% RSLogix 500 project BINSCRUBBER #49 SETTON 9-12-2016 - copy Jeff.RSS, saved by version 10.00.00.00 %
PROJECT "JBT BIN"    % processor: MicroLogix 1200 %

PROGRAM FILES
  LAD 2 "MAIN"  10 rungs
  LAD 3 "START_UP"  7 rungs
  LAD 4 "ENCODER"  11 rungs
  LAD 5 "CRADDLE"  33 rungs
  LAD 6 "BRUSH"  26 rungs
  LAD 7 "WATER"  16 rungs
  LAD 8 "AUXILARY"  14 rungs
  LAD 9 "FAULTS"  43 rungs
  LAD 10 "CONVEYORS"  16 rungs
  LAD 11 "BIN SIZING"  9 rungs

DATA FILES
  O0 OUTPUT  6 elements
  I1 INPUT  6 elements
  S2 STATUS  66 elements
  B3 BINARY  5 elements
  T4 TIMER  35 elements
  C5 COUNTER  1 elements
  R6 CONTROL  1 elements
  N7 INTEGER  34 elements
  F8 FLOAT  1 elements
  L9   1 elements
  L10   2 elements

LADDER 2 "MAIN"
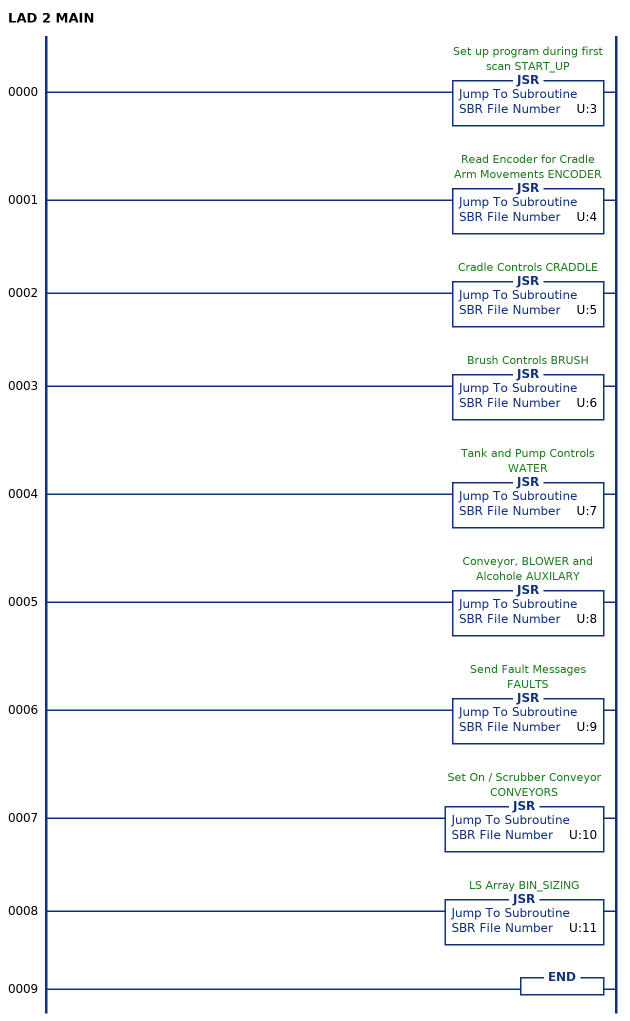
% Rung: 0 %
SOR JSR U:3 EOR
%   U:3  START_UP  "Set up program during first scan" %
% Rung: 1 %
SOR JSR U:4 EOR
%   U:4  ENCODER  "Read Encoder for Cradle Arm Movements" %
% Rung: 2 %
SOR JSR U:5 EOR
%   U:5  CRADDLE  "Cradle Controls" %
% Rung: 3 %
SOR JSR U:6 EOR
%   U:6  BRUSH  "Brush Controls" %
% Rung: 4 %
SOR JSR U:7 EOR
%   U:7  WATER  "Tank and Pump Controls" %
% Rung: 5 %
SOR JSR U:8 EOR
%   U:8  AUXILARY  "Conveyor, BLOWER and Alcohole" %
% Rung: 6 %
SOR JSR U:9 EOR
%   U:9  FAULTS  "Send Fault Messages" %
% Rung: 7 %
SOR JSR U:10 EOR
%   U:10  CONVEYORS  "Set On / Scrubber Conveyor" %
% Rung: 8 %
SOR JSR U:11 EOR
%   U:11  BIN_SIZING  "LS Array" %
% Rung: 9 %
SOR END EOR

LADDER 3 "START_UP"
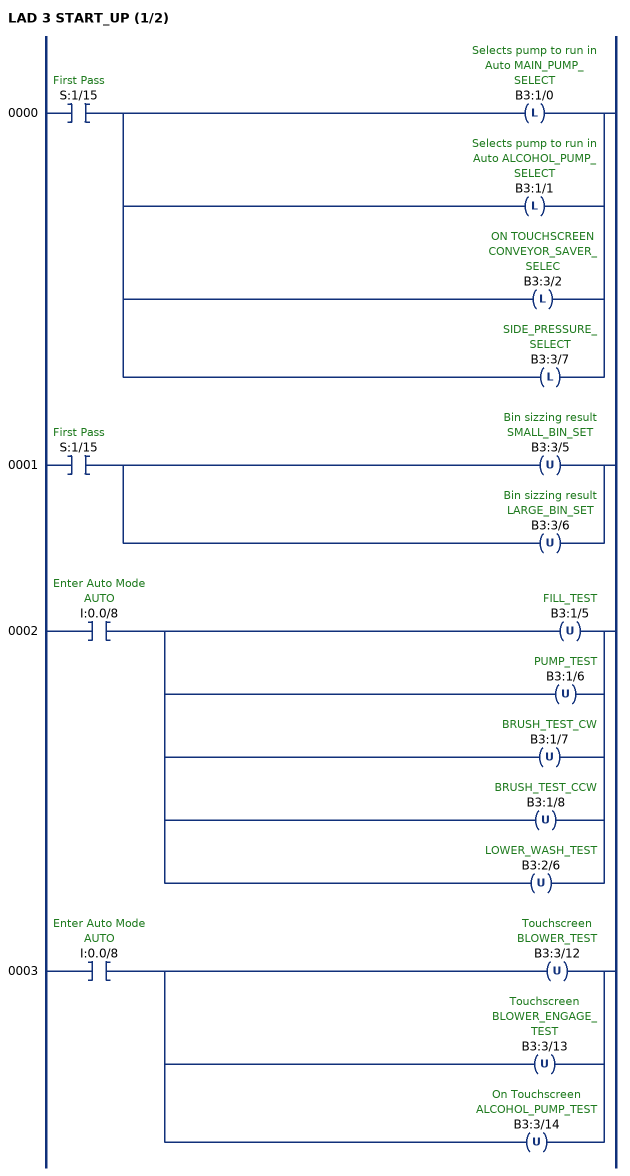
% Rung: 0 %
SOR XIC S:1/15 BST OTL B3:1/0 NXB BST OTL B3:1/1 NXB BST OTL B3:3/2 NXB OTL B3:3/7 BND BND BND EOR
%   S:1/15  "First Pass" %
%   B3:1/0  MAIN_PUMP_SELECT  "Selects pump to run in Auto" %
%   B3:1/1  ALCOHOL_PUMP_SELECT  "Selects pump to run in Auto" %
%   B3:3/2  CONVEYOR_SAVER_SELEC  "ON TOUCHSCREEN" %
%   B3:3/7  SIDE_PRESSURE_SELECT %
% Rung: 1 %
SOR XIC S:1/15 BST OTU B3:3/5 NXB OTU B3:3/6 BND EOR
%   S:1/15  "First Pass" %
%   B3:3/5  SMALL_BIN_SET  "Bin sizzing result" %
%   B3:3/6  LARGE_BIN_SET  "Bin sizzing result" %
% Rung: 2 %
SOR XIC I:0.0/8 BST OTU B3:1/5 NXB BST OTU B3:1/6 NXB OTU B3:1/7 NXB BST OTU B3:1/8 NXB OTU B3:2/6 BND BND BND EOR
%   I:0.0/8  AUTO  "Enter Auto Mode" %
%   B3:1/5  FILL_TEST %
%   B3:1/6  PUMP_TEST %
%   B3:1/7  BRUSH_TEST_CW %
%   B3:1/8  BRUSH_TEST_CCW %
%   B3:2/6  LOWER_WASH_TEST %
% Rung: 3 %
SOR XIC I:0.0/8 BST OTU B3:3/12 NXB OTU B3:3/13 NXB OTU B3:3/14 BND EOR
%   I:0.0/8  AUTO  "Enter Auto Mode" %
%   B3:3/12  BLOWER_TEST  "Touchscreen" %
%   B3:3/13  BLOWER_ENGAGE_TEST  "Touchscreen" %
%   B3:3/14  ALCOHOL_PUMP_TEST  "On Touchscreen" %

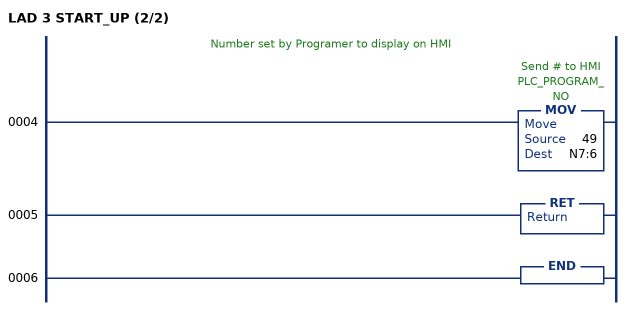
% Rung: 4 %
% Number set by Programer to display on HMI %
SOR MOV 49 N7:6 EOR
%   N7:6  PLC_PROGRAM_NO  "Send # to HMI" %
% Rung: 5 %
SOR RET EOR
% Rung: 6 %
SOR END EOR

LADDER 4 "ENCODER"
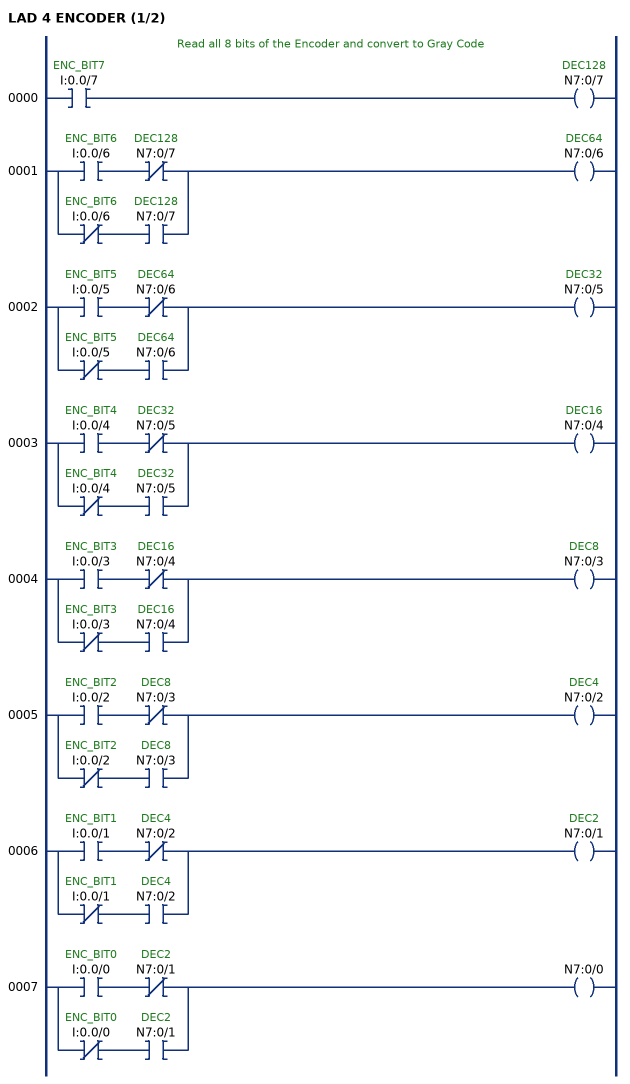
% Rung: 0 %
% Read all 8 bits of the Encoder and convert to Gray Code %
SOR XIC I:0.0/7 OTE N7:0/7 EOR
%   I:0.0/7  ENC_BIT7 %
%   N7:0/7  "DEC128" %
% Rung: 1 %
SOR BST XIC I:0.0/6 XIO N7:0/7 NXB XIO I:0.0/6 XIC N7:0/7 BND OTE N7:0/6 EOR
%   I:0.0/6  ENC_BIT6 %
%   N7:0/7  "DEC128" %
%   N7:0/6  "DEC64" %
% Rung: 2 %
SOR BST XIC I:0.0/5 XIO N7:0/6 NXB XIO I:0.0/5 XIC N7:0/6 BND OTE N7:0/5 EOR
%   I:0.0/5  ENC_BIT5 %
%   N7:0/6  "DEC64" %
%   N7:0/5  "DEC32" %
% Rung: 3 %
SOR BST XIC I:0.0/4 XIO N7:0/5 NXB XIO I:0.0/4 XIC N7:0/5 BND OTE N7:0/4 EOR
%   I:0.0/4  ENC_BIT4 %
%   N7:0/5  "DEC32" %
%   N7:0/4  "DEC16" %
% Rung: 4 %
SOR BST XIC I:0.0/3 XIO N7:0/4 NXB XIO I:0.0/3 XIC N7:0/4 BND OTE N7:0/3 EOR
%   I:0.0/3  ENC_BIT3 %
%   N7:0/4  "DEC16" %
%   N7:0/3  "DEC8" %
% Rung: 5 %
SOR BST XIC I:0.0/2 XIO N7:0/3 NXB XIO I:0.0/2 XIC N7:0/3 BND OTE N7:0/2 EOR
%   I:0.0/2  ENC_BIT2 %
%   N7:0/3  "DEC8" %
%   N7:0/2  "DEC4" %
% Rung: 6 %
SOR BST XIC I:0.0/1 XIO N7:0/2 NXB XIO I:0.0/1 XIC N7:0/2 BND OTE N7:0/1 EOR
%   I:0.0/1  ENC_BIT1 %
%   N7:0/2  "DEC4" %
%   N7:0/1  "DEC2" %
% Rung: 7 %
SOR BST XIC I:0.0/0 XIO N7:0/1 NXB XIO I:0.0/0 XIC N7:0/1 BND OTE N7:0/0 EOR
%   I:0.0/0  ENC_BIT0 %
%   N7:0/1  "DEC2" %

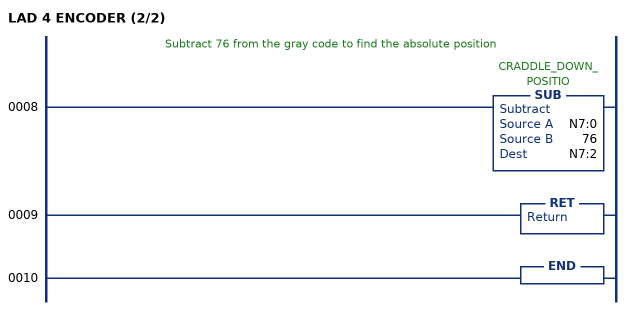
% Rung: 8 %
% Subtract 76 from the gray code to find the absolute position %
SOR SUB N7:0 76 N7:2 EOR
%   N7:0  ENC_POS %
%   N7:2  CRADDLE_DOWN_POSITIO %
% Rung: 9 %
SOR RET EOR
% Rung: 10 %
SOR END EOR

LADDER 5 "CRADDLE"
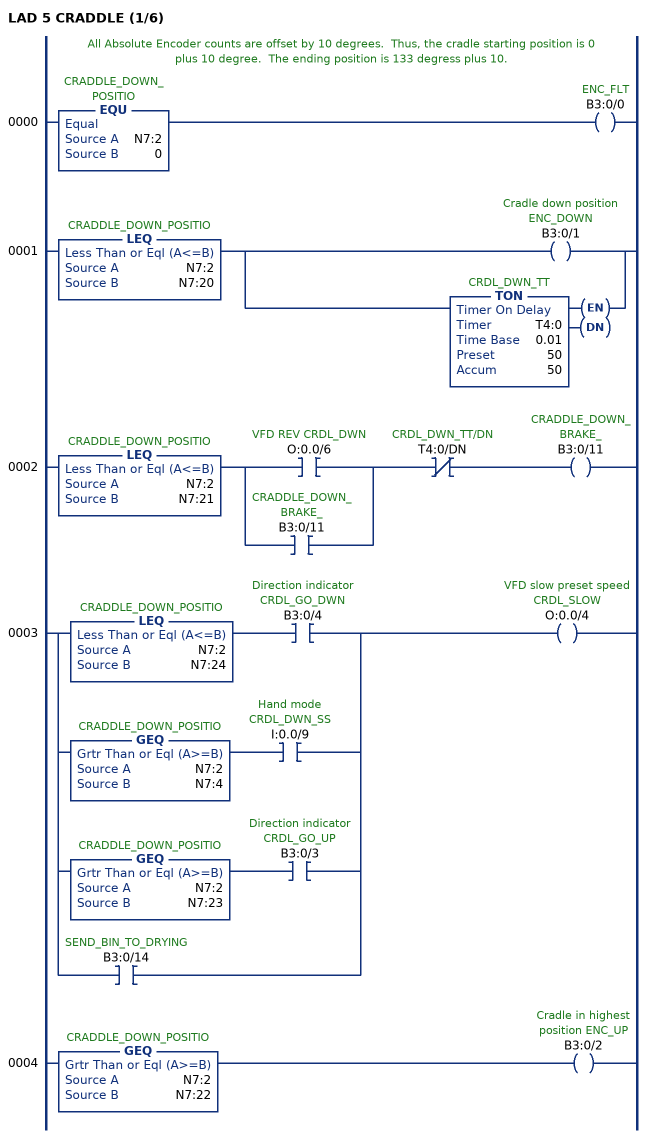
% Rung: 0 %
% All Absolute Encoder counts are offset by 10 degrees.  Thus, the cradle starting position is 0 plus 10 degree.  The ending position is 133 degress plus 10. %
SOR EQU N7:2 0 OTE B3:0/0 EOR
%   N7:2  CRADDLE_DOWN_POSITIO %
%   B3:0/0  ENC_FLT %
% Rung: 1 %
SOR LEQ N7:2 N7:20 BST OTE B3:0/1 NXB TON T4:0 0.01 50 50 BND EOR
%   N7:2  CRADDLE_DOWN_POSITIO %
%   N7:20  PICKUP_POSITION %
%   B3:0/1  ENC_DOWN  "Cradle down position" %
%   T4:0  CRDL_DWN_TT %
% Rung: 2 %
SOR LEQ N7:2 N7:21 BST XIC O:0.0/6 NXB XIC B3:0/11 BND XIO T4:0/DN OTE B3:0/11 EOR
%   N7:2  CRADDLE_DOWN_POSITIO %
%   N7:21  BRAKE_REALEASE  "Pick up position" %
%   O:0.0/6  CRDL_DWN  "VFD REV" %
%   B3:0/11  CRADDLE_DOWN_BRAKE_ %
%   T4:0  CRDL_DWN_TT %
% Rung: 3 %
SOR BST LEQ N7:2 N7:24 XIC B3:0/4 NXB GEQ N7:2 N7:4 XIC I:0.0/9 NXB BST GEQ N7:2 N7:23 XIC B3:0/3 NXB XIC B3:0/14 BND BND OTE O:0.0/4 EOR
%   N7:2  CRADDLE_DOWN_POSITIO %
%   N7:24  DOWN_SLOW_POSITION %
%   B3:0/4  CRDL_GO_DWN  "Direction indicator" %
%   N7:4  DRYING_POSITION %
%   I:0.0/9  CRDL_DWN_SS  "Hand mode" %
%   N7:23  UP_SLOW_POSITION %
%   B3:0/3  CRDL_GO_UP  "Direction indicator" %
%   B3:0/14  SEND_BIN_TO_DRYING %
%   O:0.0/4  CRDL_SLOW  "VFD slow preset speed" %
% Rung: 4 %
SOR GEQ N7:2 N7:22 OTE B3:0/2 EOR
%   N7:2  CRADDLE_DOWN_POSITIO %
%   N7:22  SCRUBBING_POSITION %
%   B3:0/2  ENC_UP  "Cradle in highest position" %

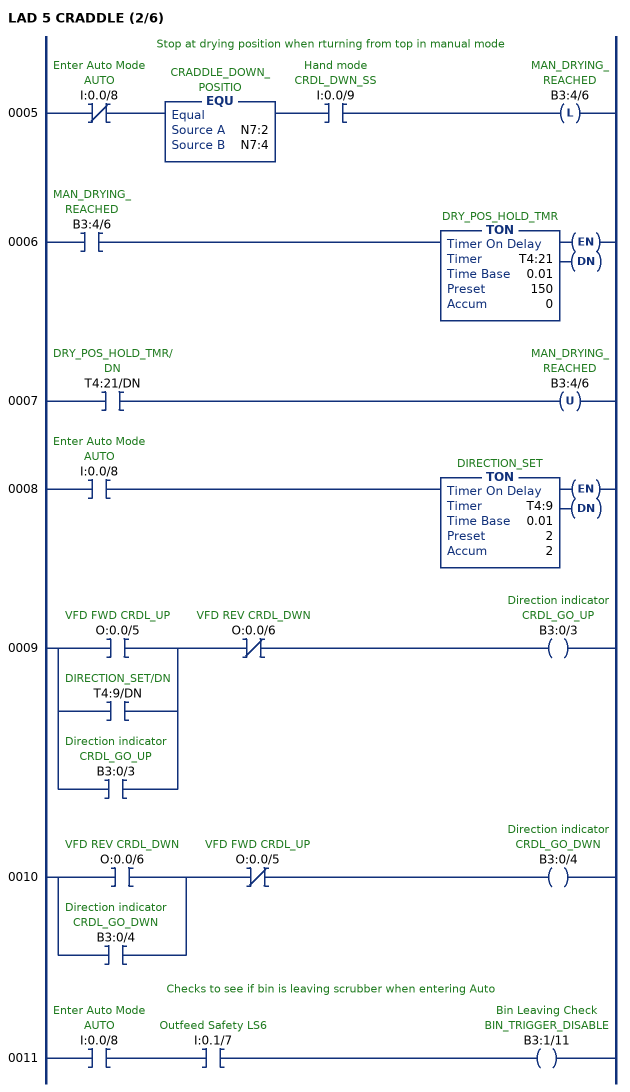
% Rung: 5 %
% Stop at drying position when rturning from top in manual mode %
SOR XIO I:0.0/8 EQU N7:2 N7:4 XIC I:0.0/9 OTL B3:4/6 EOR
%   I:0.0/8  AUTO  "Enter Auto Mode" %
%   N7:2  CRADDLE_DOWN_POSITIO %
%   N7:4  DRYING_POSITION %
%   I:0.0/9  CRDL_DWN_SS  "Hand mode" %
%   B3:4/6  MAN_DRYING_REACHED %
% Rung: 6 %
SOR XIC B3:4/6 TON T4:21 0.01 150 0 EOR
%   B3:4/6  MAN_DRYING_REACHED %
%   T4:21  DRY_POS_HOLD_TMR %
% Rung: 7 %
SOR XIC T4:21/DN OTU B3:4/6 EOR
%   T4:21  DRY_POS_HOLD_TMR %
%   B3:4/6  MAN_DRYING_REACHED %
% Rung: 8 %
SOR XIC I:0.0/8 TON T4:9 0.01 2 2 EOR
%   I:0.0/8  AUTO  "Enter Auto Mode" %
%   T4:9  DIRECTION_SET %
% Rung: 9 %
SOR BST XIC O:0.0/5 NXB XIC T4:9/DN NXB XIC B3:0/3 BND XIO O:0.0/6 OTE B3:0/3 EOR
%   O:0.0/5  CRDL_UP  "VFD FWD" %
%   T4:9  DIRECTION_SET %
%   B3:0/3  CRDL_GO_UP  "Direction indicator" %
%   O:0.0/6  CRDL_DWN  "VFD REV" %
% Rung: 10 %
SOR BST XIC O:0.0/6 NXB XIC B3:0/4 BND XIO O:0.0/5 OTE B3:0/4 EOR
%   O:0.0/6  CRDL_DWN  "VFD REV" %
%   B3:0/4  CRDL_GO_DWN  "Direction indicator" %
%   O:0.0/5  CRDL_UP  "VFD FWD" %
% Rung: 11 %
% Checks to see if bin is leaving scrubber when entering Auto %
SOR XIC I:0.0/8 XIC I:0.1/7 OTE B3:1/11 EOR
%   I:0.0/8  AUTO  "Enter Auto Mode" %
%   I:0.1/7  LS6  "Outfeed Safety" %
%   B3:1/11  BIN_TRIGGER_DISABLE  "Bin Leaving Check" %

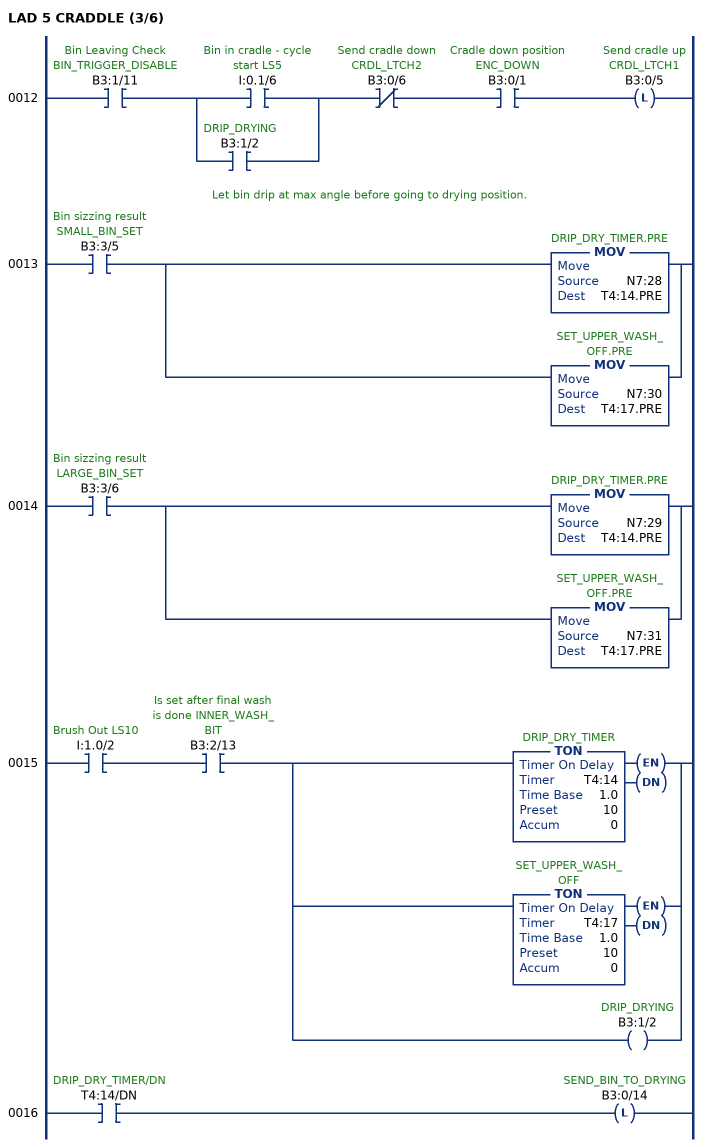
% Rung: 12 %
SOR XIC B3:1/11 BST XIC I:0.1/6 NXB XIC B3:1/2 BND XIO B3:0/6 XIC B3:0/1 OTL B3:0/5 EOR
%   B3:1/11  BIN_TRIGGER_DISABLE  "Bin Leaving Check" %
%   I:0.1/6  LS5  "Bin in cradle - cycle start" %
%   B3:1/2  DRIP_DRYING %
%   B3:0/6  CRDL_LTCH2  "Send cradle down" %
%   B3:0/1  ENC_DOWN  "Cradle down position" %
%   B3:0/5  CRDL_LTCH1  "Send cradle up" %
% Rung: 13 %
% Let bin drip at max angle before going to drying position. %
SOR XIC B3:3/5 BST MOV N7:28 T4:14.PRE NXB MOV N7:30 T4:17.PRE BND EOR
%   B3:3/5  SMALL_BIN_SET  "Bin sizzing result" %
%   N7:28  DRIP_DRY_SMALL_BIN %
%   T4:14  DRIP_DRY_TIMER %
%   N7:30  UPPER_OFF_SMALL_BIN  "TURN WASH OFF" %
%   T4:17  SET_UPPER_WASH_OFF %
% Rung: 14 %
SOR XIC B3:3/6 BST MOV N7:29 T4:14.PRE NXB MOV N7:31 T4:17.PRE BND EOR
%   B3:3/6  LARGE_BIN_SET  "Bin sizzing result" %
%   N7:29  DRIP_DRY_LARGE_BIN %
%   T4:14  DRIP_DRY_TIMER %
%   N7:31  UPPER_OFF_LARGE_BIN  "TURN WASH OFF" %
%   T4:17  SET_UPPER_WASH_OFF %
% Rung: 15 %
SOR XIC I:1.0/2 XIC B3:2/13 BST TON T4:14 1.0 10 0 NXB TON T4:17 1.0 10 0 NXB OTE B3:1/2 BND EOR
%   I:1.0/2  LS10  "Brush Out" %
%   B3:2/13  INNER_WASH_BIT  "Is set after final wash is done" %
%   T4:14  DRIP_DRY_TIMER %
%   T4:17  SET_UPPER_WASH_OFF %
%   B3:1/2  DRIP_DRYING %
% Rung: 16 %
SOR XIC T4:14/DN OTL B3:0/14 EOR
%   T4:14  DRIP_DRY_TIMER %
%   B3:0/14  SEND_BIN_TO_DRYING %

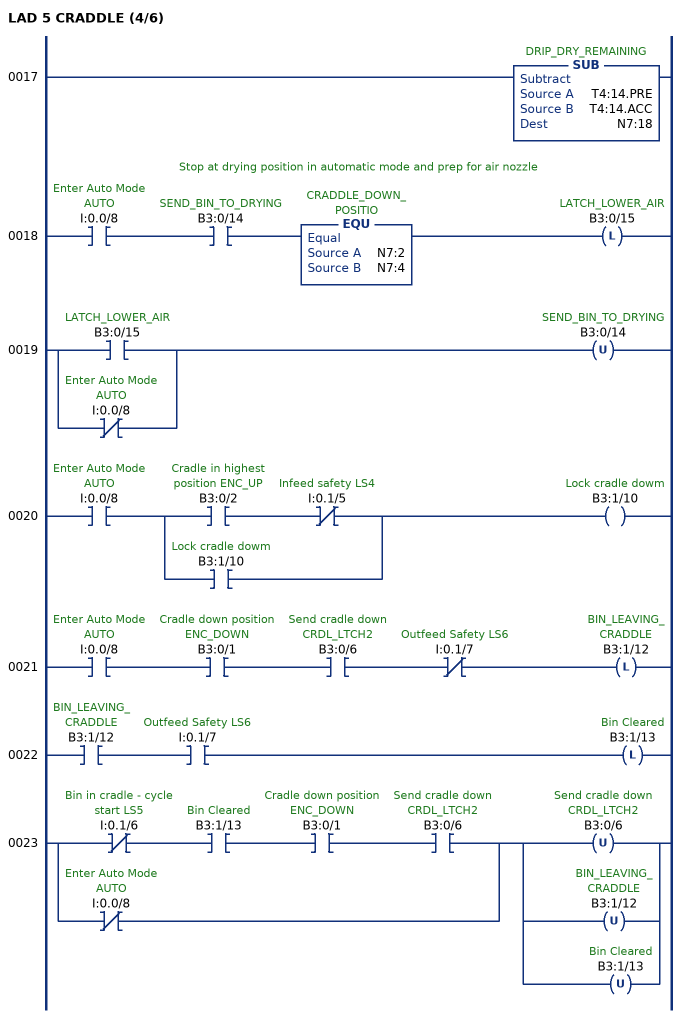
% Rung: 17 %
SOR SUB T4:14.PRE T4:14.ACC N7:18 EOR
%   T4:14  DRIP_DRY_TIMER %
%   N7:18  DRIP_DRY_REMAINING %
% Rung: 18 %
% Stop at drying position in automatic mode and prep for air nozzle %
SOR XIC I:0.0/8 XIC B3:0/14 EQU N7:2 N7:4 OTL B3:0/15 EOR
%   I:0.0/8  AUTO  "Enter Auto Mode" %
%   B3:0/14  SEND_BIN_TO_DRYING %
%   N7:2  CRADDLE_DOWN_POSITIO %
%   N7:4  DRYING_POSITION %
%   B3:0/15  LATCH_LOWER_AIR %
% Rung: 19 %
SOR BST XIC B3:0/15 NXB XIO I:0.0/8 BND OTU B3:0/14 EOR
%   B3:0/15  LATCH_LOWER_AIR %
%   I:0.0/8  AUTO  "Enter Auto Mode" %
%   B3:0/14  SEND_BIN_TO_DRYING %
% Rung: 20 %
SOR XIC I:0.0/8 BST XIC B3:0/2 XIO I:0.1/5 NXB XIC B3:1/10 BND OTE B3:1/10 EOR
%   I:0.0/8  AUTO  "Enter Auto Mode" %
%   B3:0/2  ENC_UP  "Cradle in highest position" %
%   I:0.1/5  LS4  "Infeed safety" %
%   B3:1/10  "Lock cradle dowm" %
% Rung: 21 %
SOR XIC I:0.0/8 XIC B3:0/1 XIC B3:0/6 XIO I:0.1/7 OTL B3:1/12 EOR
%   I:0.0/8  AUTO  "Enter Auto Mode" %
%   B3:0/1  ENC_DOWN  "Cradle down position" %
%   B3:0/6  CRDL_LTCH2  "Send cradle down" %
%   I:0.1/7  LS6  "Outfeed Safety" %
%   B3:1/12  BIN_LEAVING_CRADDLE %
% Rung: 22 %
SOR XIC B3:1/12 XIC I:0.1/7 OTL B3:1/13 EOR
%   B3:1/12  BIN_LEAVING_CRADDLE %
%   I:0.1/7  LS6  "Outfeed Safety" %
%   B3:1/13  "Bin Cleared" %
% Rung: 23 %
SOR BST XIO I:0.1/6 XIC B3:1/13 XIC B3:0/1 XIC B3:0/6 NXB XIO I:0.0/8 BND BST OTU B3:0/6 NXB BST OTU B3:1/12 NXB OTU B3:1/13 BND BND EOR
%   I:0.1/6  LS5  "Bin in cradle - cycle start" %
%   B3:1/13  "Bin Cleared" %
%   B3:0/1  ENC_DOWN  "Cradle down position" %
%   B3:0/6  CRDL_LTCH2  "Send cradle down" %
%   I:0.0/8  AUTO  "Enter Auto Mode" %
%   B3:1/12  BIN_LEAVING_CRADDLE %

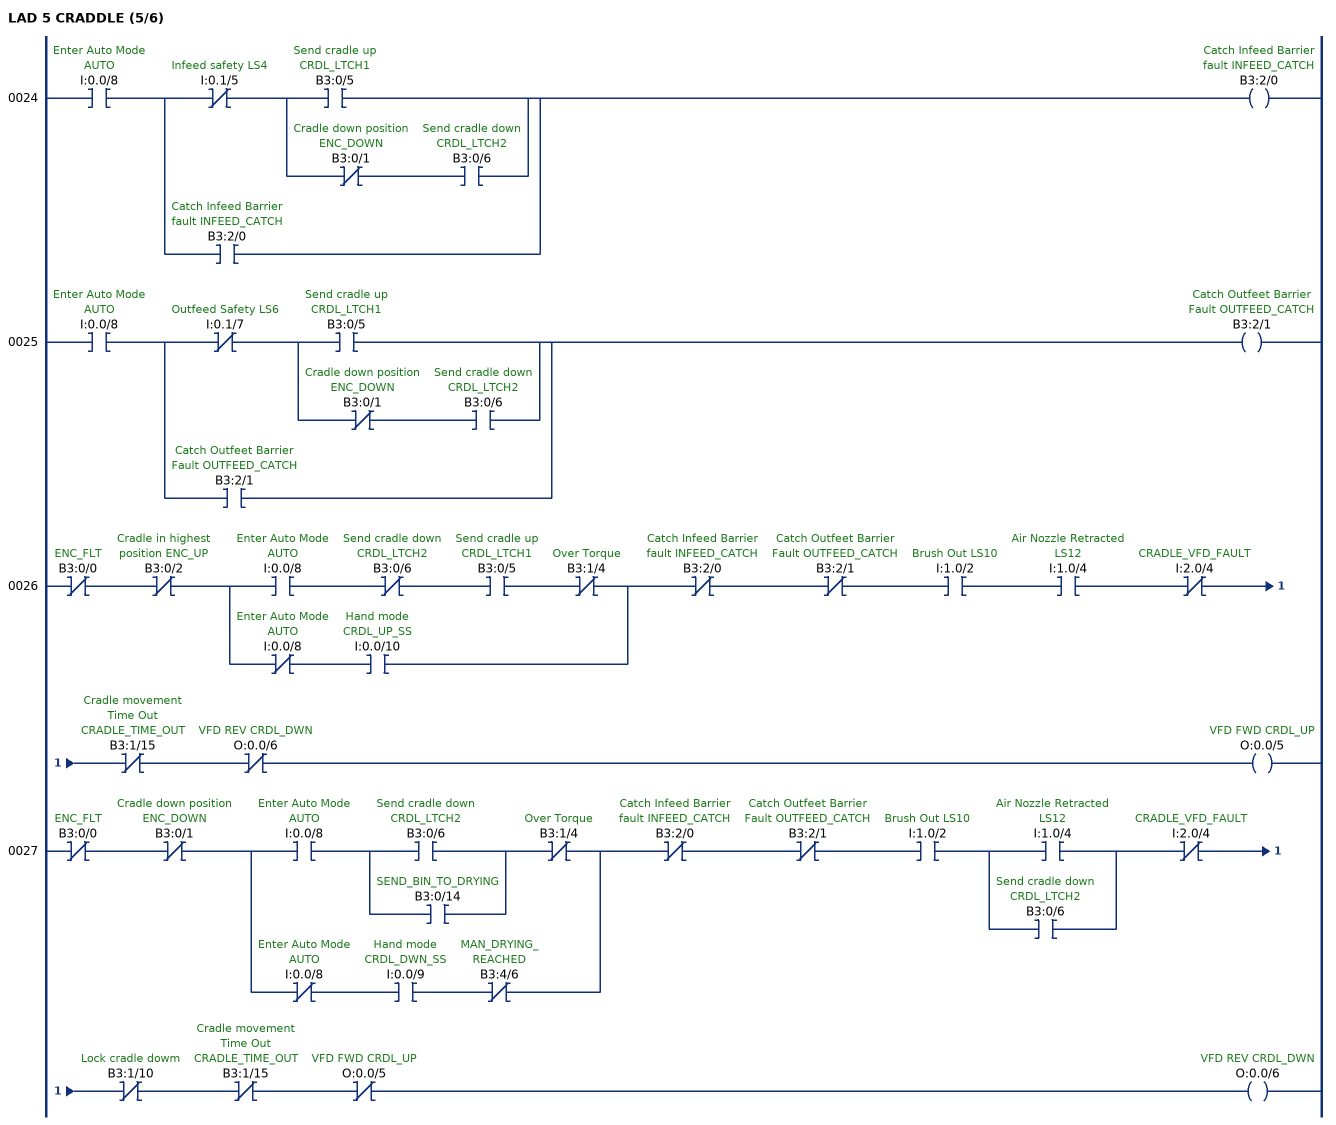
% Rung: 24 %
SOR XIC I:0.0/8 BST XIO I:0.1/5 BST XIC B3:0/5 NXB XIO B3:0/1 XIC B3:0/6 BND NXB XIC B3:2/0 BND OTE B3:2/0 EOR
%   I:0.0/8  AUTO  "Enter Auto Mode" %
%   I:0.1/5  LS4  "Infeed safety" %
%   B3:0/5  CRDL_LTCH1  "Send cradle up" %
%   B3:0/1  ENC_DOWN  "Cradle down position" %
%   B3:0/6  CRDL_LTCH2  "Send cradle down" %
%   B3:2/0  INFEED_CATCH  "Catch Infeed Barrier fault" %
% Rung: 25 %
SOR XIC I:0.0/8 BST XIO I:0.1/7 BST XIC B3:0/5 NXB XIO B3:0/1 XIC B3:0/6 BND NXB XIC B3:2/1 BND OTE B3:2/1 EOR
%   I:0.0/8  AUTO  "Enter Auto Mode" %
%   I:0.1/7  LS6  "Outfeed Safety" %
%   B3:0/5  CRDL_LTCH1  "Send cradle up" %
%   B3:0/1  ENC_DOWN  "Cradle down position" %
%   B3:0/6  CRDL_LTCH2  "Send cradle down" %
%   B3:2/1  OUTFEED_CATCH  "Catch Outfeet Barrier Fault" %
% Rung: 26 %
SOR XIO B3:0/0 XIO B3:0/2 BST XIC I:0.0/8 XIO B3:0/6 XIC B3:0/5 XIO B3:1/4 NXB XIO I:0.0/8 XIC I:0.0/10 BND XIO B3:2/0 XIO B3:2/1 XIC I:1.0/2 XIC I:1.0/4 XIO I:2.0/4 XIO B3:1/15 XIO O:0.0/6 OTE O:0.0/5 EOR
%   B3:0/0  ENC_FLT %
%   B3:0/2  ENC_UP  "Cradle in highest position" %
%   I:0.0/8  AUTO  "Enter Auto Mode" %
%   B3:0/6  CRDL_LTCH2  "Send cradle down" %
%   B3:0/5  CRDL_LTCH1  "Send cradle up" %
%   B3:1/4  "Over Torque" %
%   I:0.0/10  CRDL_UP_SS  "Hand mode" %
%   B3:2/0  INFEED_CATCH  "Catch Infeed Barrier fault" %
%   B3:2/1  OUTFEED_CATCH  "Catch Outfeet Barrier Fault" %
%   I:1.0/2  LS10  "Brush Out" %
%   I:1.0/4  LS12  "Air Nozzle Retracted" %
%   I:2.0/4  CRADLE_VFD_FAULT %
%   B3:1/15  CRADLE_TIME_OUT  "Cradle movement Time Out" %
%   O:0.0/6  CRDL_DWN  "VFD REV" %
%   O:0.0/5  CRDL_UP  "VFD FWD" %
% Rung: 27 %
SOR XIO B3:0/0 XIO B3:0/1 BST XIC I:0.0/8 BST XIC B3:0/6 NXB XIC B3:0/14 BND XIO B3:1/4 NXB XIO I:0.0/8 XIC I:0.0/9 XIO B3:4/6 BND XIO B3:2/0 XIO B3:2/1 XIC I:1.0/2 BST XIC I:1.0/4 NXB XIC B3:0/6 BND XIO I:2.0/4 XIO B3:1/10 XIO B3:1/15 XIO O:0.0/5 OTE O:0.0/6 EOR
%   B3:0/0  ENC_FLT %
%   B3:0/1  ENC_DOWN  "Cradle down position" %
%   I:0.0/8  AUTO  "Enter Auto Mode" %
%   B3:0/6  CRDL_LTCH2  "Send cradle down" %
%   B3:0/14  SEND_BIN_TO_DRYING %
%   B3:1/4  "Over Torque" %
%   I:0.0/9  CRDL_DWN_SS  "Hand mode" %
%   B3:4/6  MAN_DRYING_REACHED %
%   B3:2/0  INFEED_CATCH  "Catch Infeed Barrier fault" %
%   B3:2/1  OUTFEED_CATCH  "Catch Outfeet Barrier Fault" %
%   I:1.0/2  LS10  "Brush Out" %
%   I:1.0/4  LS12  "Air Nozzle Retracted" %
%   I:2.0/4  CRADLE_VFD_FAULT %
%   B3:1/10  "Lock cradle dowm" %
%   B3:1/15  CRADLE_TIME_OUT  "Cradle movement Time Out" %
%   O:0.0/5  CRDL_UP  "VFD FWD" %
%   O:0.0/6  CRDL_DWN  "VFD REV" %

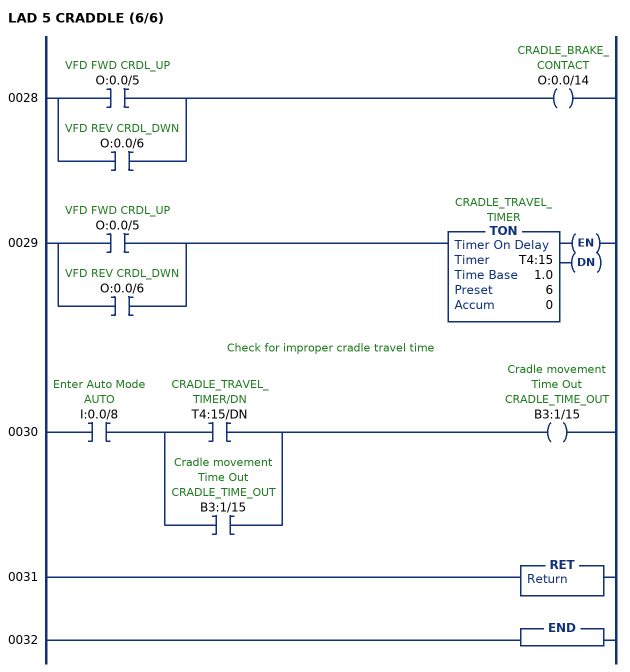
% Rung: 28 %
SOR BST XIC O:0.0/5 NXB XIC O:0.0/6 BND OTE O:0.0/14 EOR
%   O:0.0/5  CRDL_UP  "VFD FWD" %
%   O:0.0/6  CRDL_DWN  "VFD REV" %
%   O:0.0/14  CRADLE_BRAKE_CONTACT %
% Rung: 29 %
SOR BST XIC O:0.0/5 NXB XIC O:0.0/6 BND TON T4:15 1.0 6 0 EOR
%   O:0.0/5  CRDL_UP  "VFD FWD" %
%   O:0.0/6  CRDL_DWN  "VFD REV" %
%   T4:15  CRADLE_TRAVEL_TIMER %
% Rung: 30 %
% Check for improper cradle travel time %
SOR XIC I:0.0/8 BST XIC T4:15/DN NXB XIC B3:1/15 BND OTE B3:1/15 EOR
%   I:0.0/8  AUTO  "Enter Auto Mode" %
%   T4:15  CRADLE_TRAVEL_TIMER %
%   B3:1/15  CRADLE_TIME_OUT  "Cradle movement Time Out" %
% Rung: 31 %
SOR RET EOR
% Rung: 32 %
SOR END EOR

LADDER 6 "BRUSH"
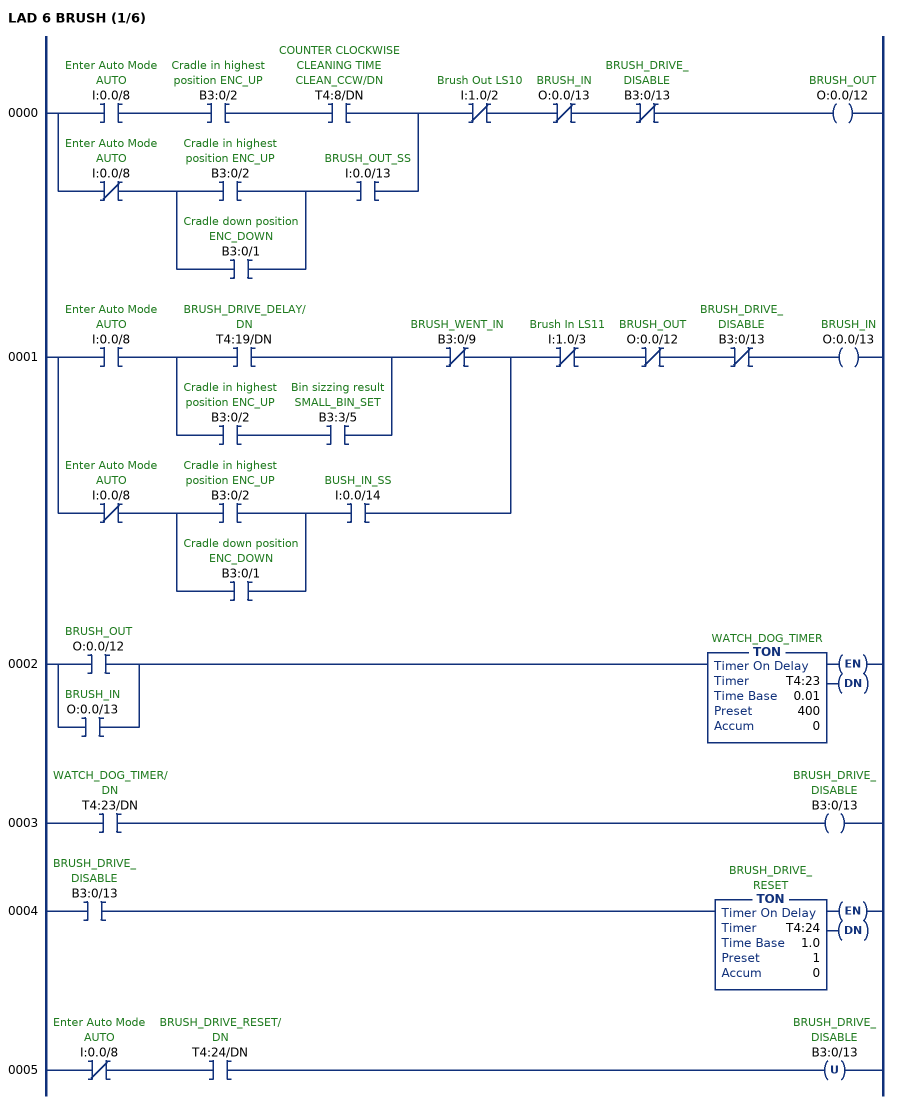
% Rung: 0 %
SOR BST XIC I:0.0/8 XIC B3:0/2 XIC T4:8/DN NXB XIO I:0.0/8 BST XIC B3:0/2 NXB XIC B3:0/1 BND XIC I:0.0/13 BND XIO I:1.0/2 XIO O:0.0/13 XIO B3:0/13 OTE O:0.0/12 EOR
%   I:0.0/8  AUTO  "Enter Auto Mode" %
%   B3:0/2  ENC_UP  "Cradle in highest position" %
%   T4:8  CLEAN_CCW  "COUNTER CLOCKWISE CLEANING TIME" %
%   B3:0/1  ENC_DOWN  "Cradle down position" %
%   I:0.0/13  BRUSH_OUT_SS %
%   I:1.0/2  LS10  "Brush Out" %
%   O:0.0/13  BRUSH_IN %
%   B3:0/13  BRUSH_DRIVE_DISABLE %
%   O:0.0/12  BRUSH_OUT %
% Rung: 1 %
SOR BST XIC I:0.0/8 BST XIC T4:19/DN NXB XIC B3:0/2 XIC B3:3/5 BND XIO B3:0/9 NXB XIO I:0.0/8 BST XIC B3:0/2 NXB XIC B3:0/1 BND XIC I:0.0/14 BND XIO I:1.0/3 XIO O:0.0/12 XIO B3:0/13 OTE O:0.0/13 EOR
%   I:0.0/8  AUTO  "Enter Auto Mode" %
%   T4:19  BRUSH_DRIVE_DELAY %
%   B3:0/2  ENC_UP  "Cradle in highest position" %
%   B3:3/5  SMALL_BIN_SET  "Bin sizzing result" %
%   B3:0/9  BRUSH_WENT_IN %
%   B3:0/1  ENC_DOWN  "Cradle down position" %
%   I:0.0/14  BUSH_IN_SS %
%   I:1.0/3  LS11  "Brush In" %
%   O:0.0/12  BRUSH_OUT %
%   B3:0/13  BRUSH_DRIVE_DISABLE %
%   O:0.0/13  BRUSH_IN %
% Rung: 2 %
SOR BST XIC O:0.0/12 NXB XIC O:0.0/13 BND TON T4:23 0.01 400 0 EOR
%   O:0.0/12  BRUSH_OUT %
%   O:0.0/13  BRUSH_IN %
%   T4:23  WATCH_DOG_TIMER %
% Rung: 3 %
SOR XIC T4:23/DN OTE B3:0/13 EOR
%   T4:23  WATCH_DOG_TIMER %
%   B3:0/13  BRUSH_DRIVE_DISABLE %
% Rung: 4 %
SOR XIC B3:0/13 TON T4:24 1.0 1 0 EOR
%   B3:0/13  BRUSH_DRIVE_DISABLE %
%   T4:24  BRUSH_DRIVE_RESET %
% Rung: 5 %
SOR XIO I:0.0/8 XIC T4:24/DN OTU B3:0/13 EOR
%   I:0.0/8  AUTO  "Enter Auto Mode" %
%   T4:24  BRUSH_DRIVE_RESET %
%   B3:0/13  BRUSH_DRIVE_DISABLE %

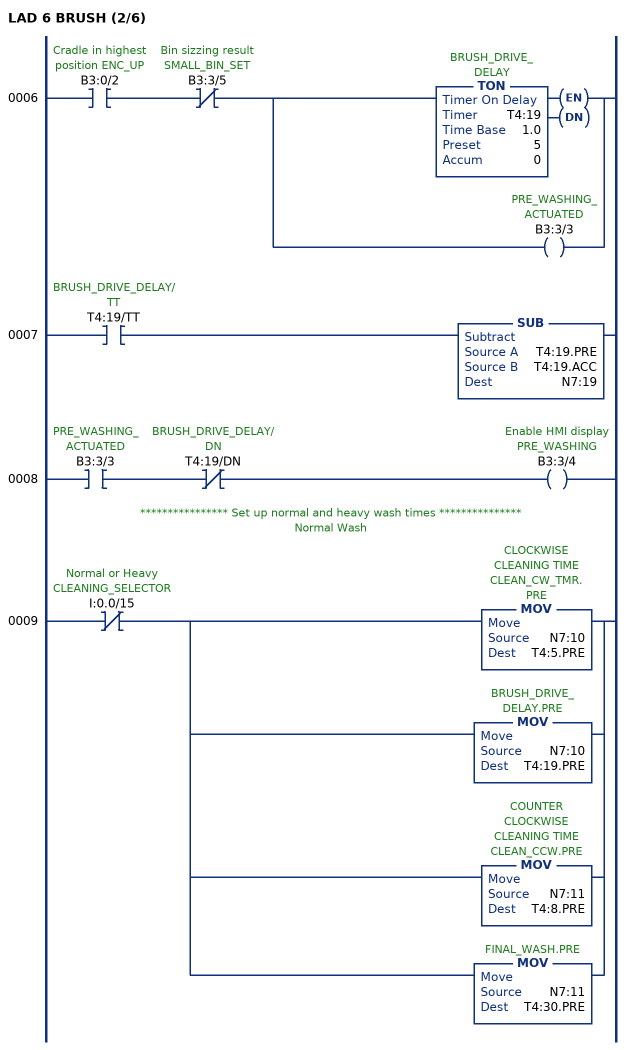
% Rung: 6 %
SOR XIC B3:0/2 XIO B3:3/5 BST TON T4:19 1.0 5 0 NXB OTE B3:3/3 BND EOR
%   B3:0/2  ENC_UP  "Cradle in highest position" %
%   B3:3/5  SMALL_BIN_SET  "Bin sizzing result" %
%   T4:19  BRUSH_DRIVE_DELAY %
%   B3:3/3  PRE_WASHING_ACTUATED %
% Rung: 7 %
SOR XIC T4:19/TT SUB T4:19.PRE T4:19.ACC N7:19 EOR
%   T4:19  BRUSH_DRIVE_DELAY %
% Rung: 8 %
SOR XIC B3:3/3 XIO T4:19/DN OTE B3:3/4 EOR
%   B3:3/3  PRE_WASHING_ACTUATED %
%   T4:19  BRUSH_DRIVE_DELAY %
%   B3:3/4  PRE_WASHING  "Enable HMI display" %
% Rung: 9 %
% **************** Set up normal and heavy wash times ***************
% Normal Wash %
SOR XIO I:0.0/15 BST MOV N7:10 T4:5.PRE NXB MOV N7:10 T4:19.PRE NXB MOV N7:11 T4:8.PRE NXB MOV N7:11 T4:30.PRE BND EOR
%   I:0.0/15  CLEANING_SELECTOR  "Normal or Heavy" %
%   N7:10  NORMAL_CW_CLEAN_TIME %
%   T4:5  CLEAN_CW_TMR  "CLOCKWISE CLEANING TIME" %
%   T4:19  BRUSH_DRIVE_DELAY %
%   N7:11  NORMAL_CCW_CLEAN_TIM %
%   T4:8  CLEAN_CCW  "COUNTER CLOCKWISE CLEANING TIME" %
%   T4:30  FINAL_WASH %

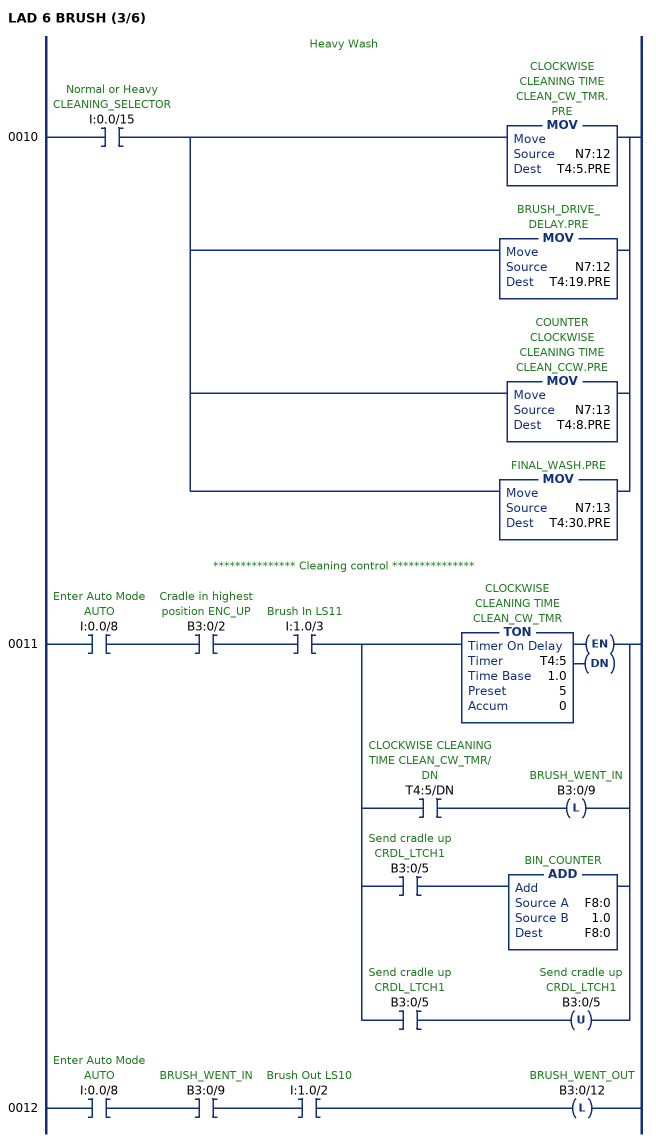
% Rung: 10 %
% Heavy Wash %
SOR XIC I:0.0/15 BST MOV N7:12 T4:5.PRE NXB MOV N7:12 T4:19.PRE NXB MOV N7:13 T4:8.PRE NXB MOV N7:13 T4:30.PRE BND EOR
%   I:0.0/15  CLEANING_SELECTOR  "Normal or Heavy" %
%   N7:12  HEAVY_CW_CLEAN_TIME %
%   T4:5  CLEAN_CW_TMR  "CLOCKWISE CLEANING TIME" %
%   T4:19  BRUSH_DRIVE_DELAY %
%   N7:13  HEAVY_CCW_CLEAN_TIME %
%   T4:8  CLEAN_CCW  "COUNTER CLOCKWISE CLEANING TIME" %
%   T4:30  FINAL_WASH %
% Rung: 11 %
% *************** Cleaning control *************** %
SOR XIC I:0.0/8 XIC B3:0/2 XIC I:1.0/3 BST TON T4:5 1.0 5 0 NXB XIC T4:5/DN OTL B3:0/9 NXB BST XIC B3:0/5 ADD F8:0 1.0 F8:0 NXB XIC B3:0/5 OTU B3:0/5 BND BND EOR
%   I:0.0/8  AUTO  "Enter Auto Mode" %
%   B3:0/2  ENC_UP  "Cradle in highest position" %
%   I:1.0/3  LS11  "Brush In" %
%   T4:5  CLEAN_CW_TMR  "CLOCKWISE CLEANING TIME" %
%   B3:0/9  BRUSH_WENT_IN %
%   B3:0/5  CRDL_LTCH1  "Send cradle up" %
%   F8:0  BIN_COUNTER %
% Rung: 12 %
SOR XIC I:0.0/8 XIC B3:0/9 XIC I:1.0/2 OTL B3:0/12 EOR
%   I:0.0/8  AUTO  "Enter Auto Mode" %
%   B3:0/9  BRUSH_WENT_IN %
%   I:1.0/2  LS10  "Brush Out" %
%   B3:0/12  BRUSH_WENT_OUT %

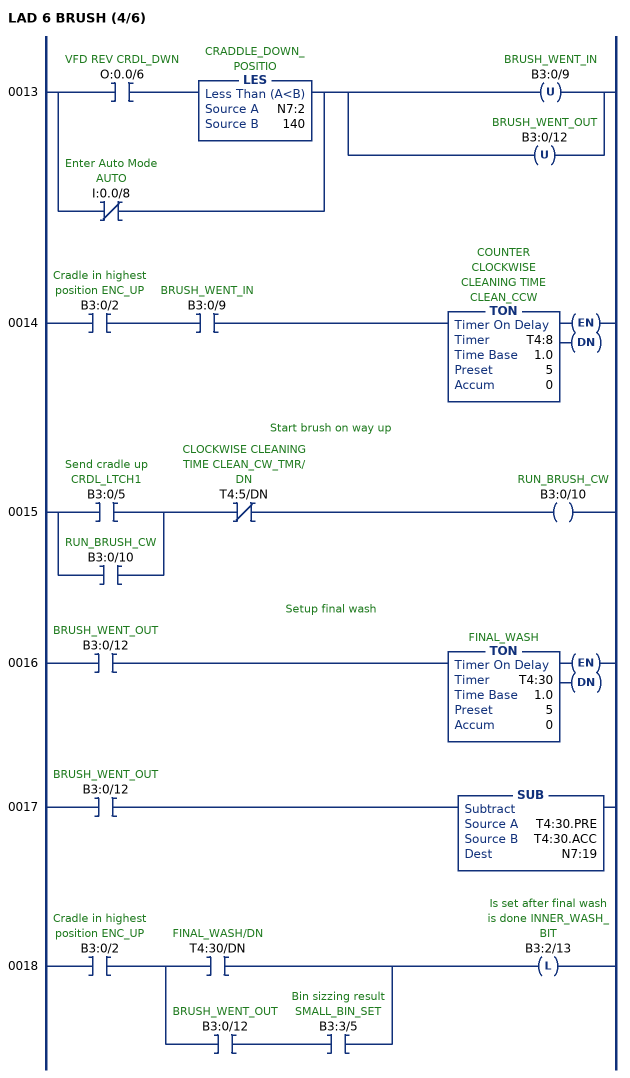
% Rung: 13 %
SOR BST XIC O:0.0/6 LES N7:2 140 NXB XIO I:0.0/8 BND BST OTU B3:0/9 NXB OTU B3:0/12 BND EOR
%   O:0.0/6  CRDL_DWN  "VFD REV" %
%   N7:2  CRADDLE_DOWN_POSITIO %
%   I:0.0/8  AUTO  "Enter Auto Mode" %
%   B3:0/9  BRUSH_WENT_IN %
%   B3:0/12  BRUSH_WENT_OUT %
% Rung: 14 %
SOR XIC B3:0/2 XIC B3:0/9 TON T4:8 1.0 5 0 EOR
%   B3:0/2  ENC_UP  "Cradle in highest position" %
%   B3:0/9  BRUSH_WENT_IN %
%   T4:8  CLEAN_CCW  "COUNTER CLOCKWISE CLEANING TIME" %
% Rung: 15 %
% Start brush on way up %
SOR BST XIC B3:0/5 NXB XIC B3:0/10 BND XIO T4:5/DN OTE B3:0/10 EOR
%   B3:0/5  CRDL_LTCH1  "Send cradle up" %
%   B3:0/10  RUN_BRUSH_CW %
%   T4:5  CLEAN_CW_TMR  "CLOCKWISE CLEANING TIME" %
% Rung: 16 %
% Setup final wash %
SOR XIC B3:0/12 TON T4:30 1.0 5 0 EOR
%   B3:0/12  BRUSH_WENT_OUT %
%   T4:30  FINAL_WASH %
% Rung: 17 %
SOR XIC B3:0/12 SUB T4:30.PRE T4:30.ACC N7:19 EOR
%   B3:0/12  BRUSH_WENT_OUT %
%   T4:30  FINAL_WASH %
% Rung: 18 %
SOR XIC B3:0/2 BST XIC T4:30/DN NXB XIC B3:0/12 XIC B3:3/5 BND OTL B3:2/13 EOR
%   B3:0/2  ENC_UP  "Cradle in highest position" %
%   T4:30  FINAL_WASH %
%   B3:0/12  BRUSH_WENT_OUT %
%   B3:3/5  SMALL_BIN_SET  "Bin sizzing result" %
%   B3:2/13  INNER_WASH_BIT  "Is set after final wash is done" %

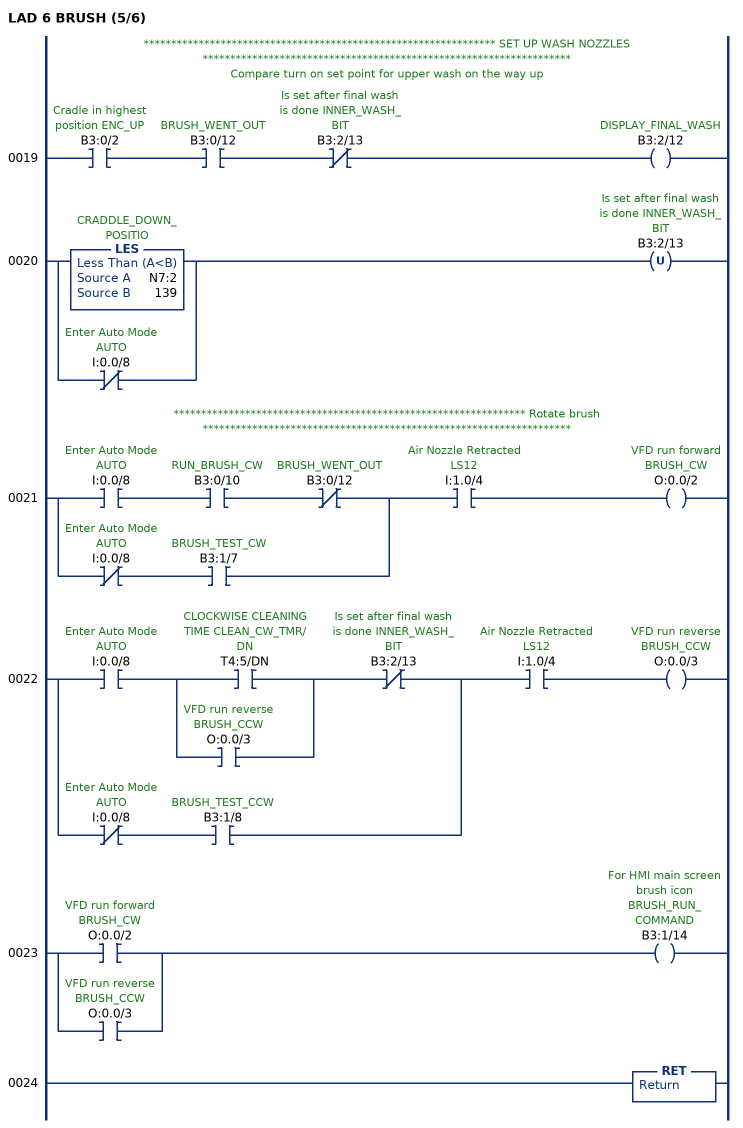
% Rung: 19 %
% **************************************************************** SET UP WASH NOZZLES  *******************************************************************
% Compare turn on set point for upper wash on the way up %
SOR XIC B3:0/2 XIC B3:0/12 XIO B3:2/13 OTE B3:2/12 EOR
%   B3:0/2  ENC_UP  "Cradle in highest position" %
%   B3:0/12  BRUSH_WENT_OUT %
%   B3:2/13  INNER_WASH_BIT  "Is set after final wash is done" %
%   B3:2/12  DISPLAY_FINAL_WASH %
% Rung: 20 %
SOR BST LES N7:2 139 NXB XIO I:0.0/8 BND OTU B3:2/13 EOR
%   N7:2  CRADDLE_DOWN_POSITIO %
%   I:0.0/8  AUTO  "Enter Auto Mode" %
%   B3:2/13  INNER_WASH_BIT  "Is set after final wash is done" %
% Rung: 21 %
% **************************************************************** Rotate brush  ******************************************************************* %
SOR BST XIC I:0.0/8 XIC B3:0/10 XIO B3:0/12 NXB XIO I:0.0/8 XIC B3:1/7 BND XIC I:1.0/4 OTE O:0.0/2 EOR
%   I:0.0/8  AUTO  "Enter Auto Mode" %
%   B3:0/10  RUN_BRUSH_CW %
%   B3:0/12  BRUSH_WENT_OUT %
%   B3:1/7  BRUSH_TEST_CW %
%   I:1.0/4  LS12  "Air Nozzle Retracted" %
%   O:0.0/2  BRUSH_CW  "VFD run forward" %
% Rung: 22 %
SOR BST XIC I:0.0/8 BST XIC T4:5/DN NXB XIC O:0.0/3 BND XIO B3:2/13 NXB XIO I:0.0/8 XIC B3:1/8 BND XIC I:1.0/4 OTE O:0.0/3 EOR
%   I:0.0/8  AUTO  "Enter Auto Mode" %
%   T4:5  CLEAN_CW_TMR  "CLOCKWISE CLEANING TIME" %
%   O:0.0/3  BRUSH_CCW  "VFD run reverse" %
%   B3:2/13  INNER_WASH_BIT  "Is set after final wash is done" %
%   B3:1/8  BRUSH_TEST_CCW %
%   I:1.0/4  LS12  "Air Nozzle Retracted" %
% Rung: 23 %
SOR BST XIC O:0.0/2 NXB XIC O:0.0/3 BND OTE B3:1/14 EOR
%   O:0.0/2  BRUSH_CW  "VFD run forward" %
%   O:0.0/3  BRUSH_CCW  "VFD run reverse" %
%   B3:1/14  BRUSH_RUN_COMMAND  "For HMI main screen brush icon" %
% Rung: 24 %
SOR RET EOR

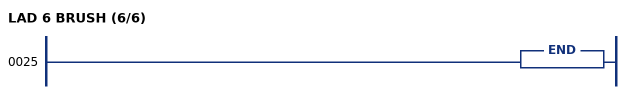
% Rung: 25 %
SOR END EOR

LADDER 7 "WATER"
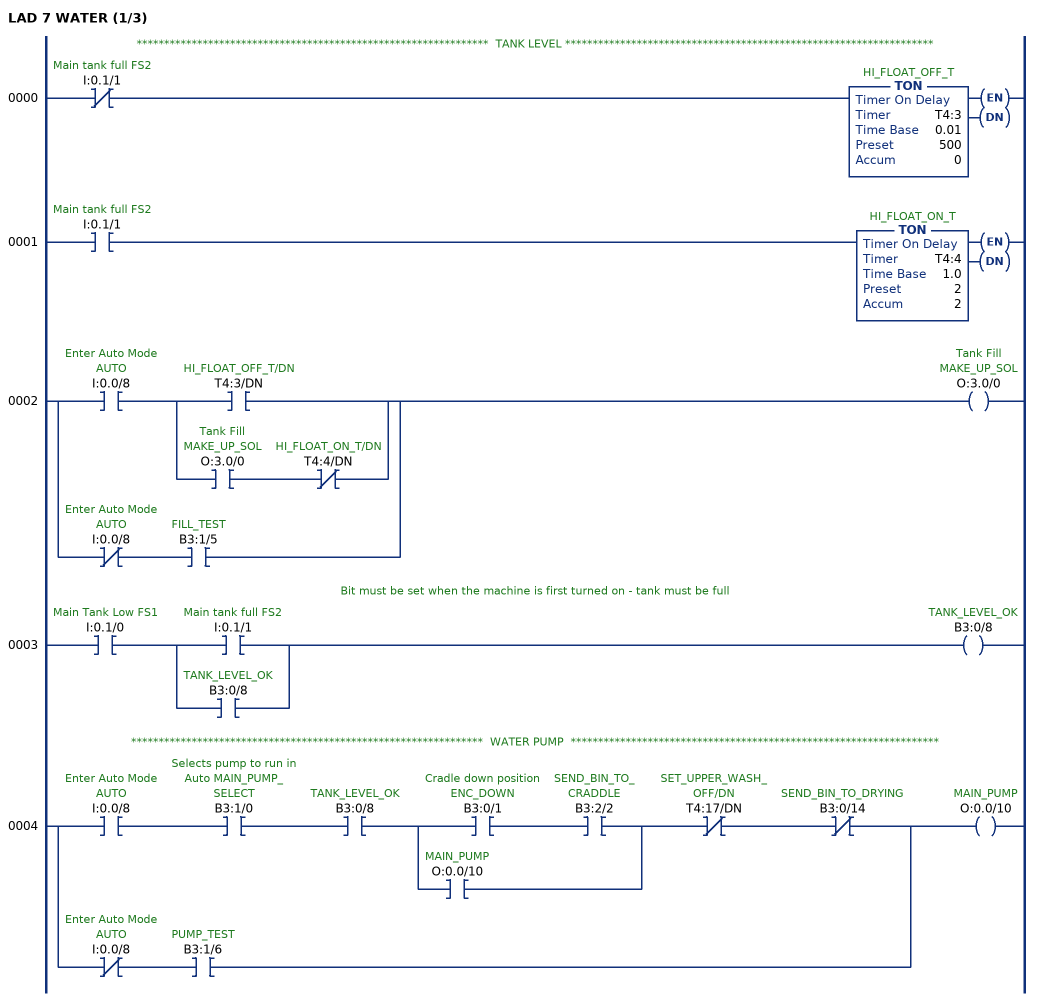
% Rung: 0 %
% ****************************************************************  TANK LEVEL ******************************************************************* %
SOR XIO I:0.1/1 TON T4:3 0.01 500 0 EOR
%   I:0.1/1  FS2  "Main tank full" %
%   T4:3  HI_FLOAT_OFF_T %
% Rung: 1 %
SOR XIC I:0.1/1 TON T4:4 1.0 2 2 EOR
%   I:0.1/1  FS2  "Main tank full" %
%   T4:4  HI_FLOAT_ON_T %
% Rung: 2 %
SOR BST XIC I:0.0/8 BST XIC T4:3/DN NXB XIC O:3.0/0 XIO T4:4/DN BND NXB XIO I:0.0/8 XIC B3:1/5 BND OTE O:3.0/0 EOR
%   I:0.0/8  AUTO  "Enter Auto Mode" %
%   T4:3  HI_FLOAT_OFF_T %
%   O:3.0/0  MAKE_UP_SOL  "Tank Fill" %
%   T4:4  HI_FLOAT_ON_T %
%   B3:1/5  FILL_TEST %
% Rung: 3 %
% Bit must be set when the machine is first turned on - tank must be full %
SOR XIC I:0.1/0 BST XIC I:0.1/1 NXB XIC B3:0/8 BND OTE B3:0/8 EOR
%   I:0.1/0  FS1  "Main Tank Low" %
%   I:0.1/1  FS2  "Main tank full" %
%   B3:0/8  TANK_LEVEL_OK %
% Rung: 4 %
% ****************************************************************  WATER PUMP  ******************************************************************* %
SOR BST XIC I:0.0/8 XIC B3:1/0 XIC B3:0/8 BST XIC B3:0/1 XIC B3:2/2 NXB XIC O:0.0/10 BND XIO T4:17/DN XIO B3:0/14 NXB XIO I:0.0/8 XIC B3:1/6 BND OTE O:0.0/10 EOR
%   I:0.0/8  AUTO  "Enter Auto Mode" %
%   B3:1/0  MAIN_PUMP_SELECT  "Selects pump to run in Auto" %
%   B3:0/8  TANK_LEVEL_OK %
%   B3:0/1  ENC_DOWN  "Cradle down position" %
%   B3:2/2  SEND_BIN_TO_CRADDLE %
%   O:0.0/10  MAIN_PUMP %
%   T4:17  SET_UPPER_WASH_OFF %
%   B3:0/14  SEND_BIN_TO_DRYING %
%   B3:1/6  PUMP_TEST %

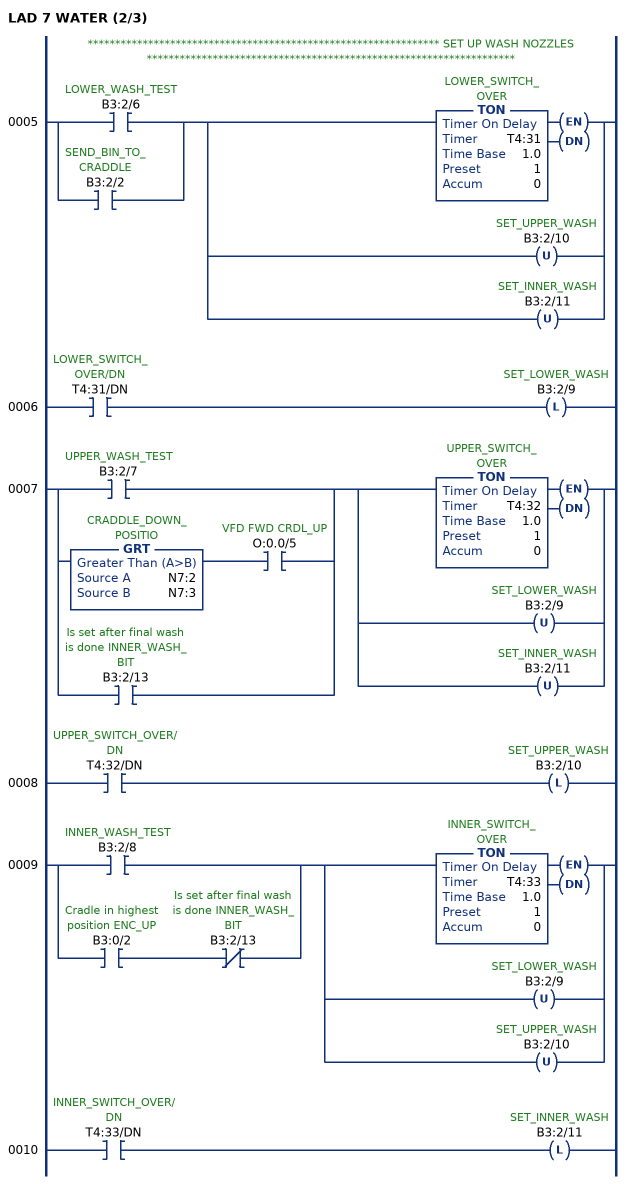
% Rung: 5 %
% **************************************************************** SET UP WASH NOZZLES  ******************************************************************* %
SOR BST XIC B3:2/6 NXB XIC B3:2/2 BND BST TON T4:31 1.0 1 0 NXB BST OTU B3:2/10 NXB OTU B3:2/11 BND BND EOR
%   B3:2/6  LOWER_WASH_TEST %
%   B3:2/2  SEND_BIN_TO_CRADDLE %
%   T4:31  LOWER_SWITCH_OVER %
%   B3:2/10  SET_UPPER_WASH %
%   B3:2/11  SET_INNER_WASH %
% Rung: 6 %
SOR XIC T4:31/DN OTL B3:2/9 EOR
%   T4:31  LOWER_SWITCH_OVER %
%   B3:2/9  SET_LOWER_WASH %
% Rung: 7 %
SOR BST BST XIC B3:2/7 NXB GRT N7:2 N7:3 XIC O:0.0/5 BND NXB XIC B3:2/13 BND BST TON T4:32 1.0 1 0 NXB BST OTU B3:2/9 NXB OTU B3:2/11 BND BND EOR
%   B3:2/7  UPPER_WASH_TEST %
%   N7:2  CRADDLE_DOWN_POSITIO %
%   N7:3  UPPER_WASH_TURN_ON %
%   O:0.0/5  CRDL_UP  "VFD FWD" %
%   B3:2/13  INNER_WASH_BIT  "Is set after final wash is done" %
%   T4:32  UPPER_SWITCH_OVER %
%   B3:2/9  SET_LOWER_WASH %
%   B3:2/11  SET_INNER_WASH %
% Rung: 8 %
SOR XIC T4:32/DN OTL B3:2/10 EOR
%   T4:32  UPPER_SWITCH_OVER %
%   B3:2/10  SET_UPPER_WASH %
% Rung: 9 %
SOR BST XIC B3:2/8 NXB XIC B3:0/2 XIO B3:2/13 BND BST TON T4:33 1.0 1 0 NXB BST OTU B3:2/9 NXB OTU B3:2/10 BND BND EOR
%   B3:2/8  INNER_WASH_TEST %
%   B3:0/2  ENC_UP  "Cradle in highest position" %
%   B3:2/13  INNER_WASH_BIT  "Is set after final wash is done" %
%   T4:33  INNER_SWITCH_OVER %
%   B3:2/9  SET_LOWER_WASH %
%   B3:2/10  SET_UPPER_WASH %
% Rung: 10 %
SOR XIC T4:33/DN OTL B3:2/11 EOR
%   T4:33  INNER_SWITCH_OVER %
%   B3:2/11  SET_INNER_WASH %

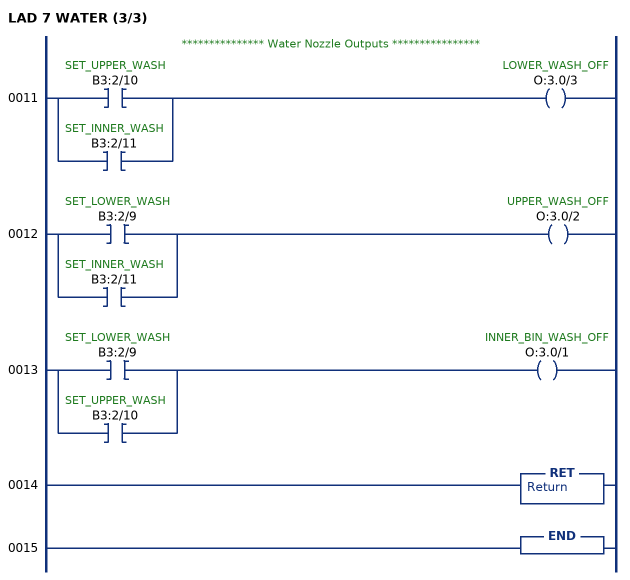
% Rung: 11 %
% *************** Water Nozzle Outputs **************** %
SOR BST XIC B3:2/10 NXB XIC B3:2/11 BND OTE O:3.0/3 EOR
%   B3:2/10  SET_UPPER_WASH %
%   B3:2/11  SET_INNER_WASH %
%   O:3.0/3  LOWER_WASH_OFF %
% Rung: 12 %
SOR BST XIC B3:2/9 NXB XIC B3:2/11 BND OTE O:3.0/2 EOR
%   B3:2/9  SET_LOWER_WASH %
%   B3:2/11  SET_INNER_WASH %
%   O:3.0/2  UPPER_WASH_OFF %
% Rung: 13 %
SOR BST XIC B3:2/9 NXB XIC B3:2/10 BND OTE O:3.0/1 EOR
%   B3:2/9  SET_LOWER_WASH %
%   B3:2/10  SET_UPPER_WASH %
%   O:3.0/1  INNER_BIN_WASH_OFF %
% Rung: 14 %
SOR RET EOR
% Rung: 15 %
SOR END EOR

LADDER 8 "AUXILARY"
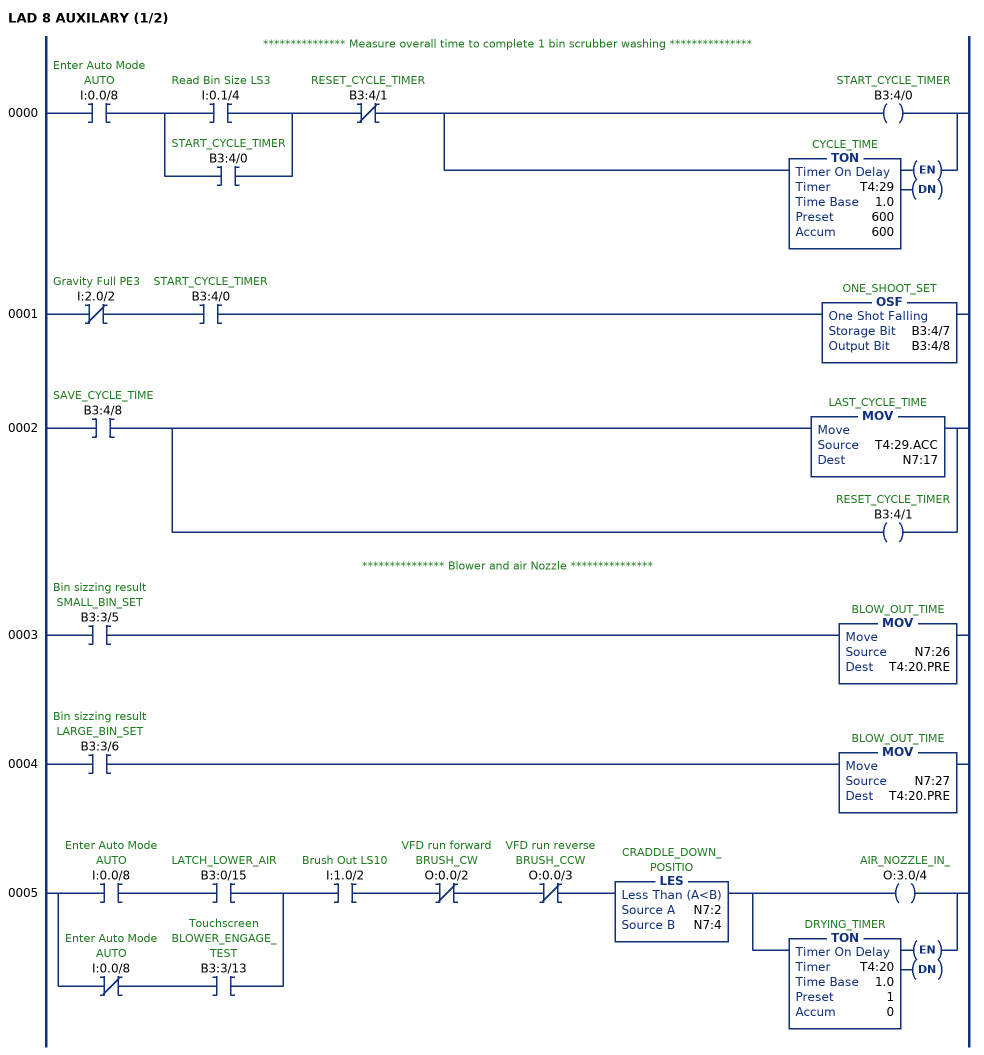
% Rung: 0 %
% *************** Measure overall time to complete 1 bin scrubber washing *************** %
SOR XIC I:0.0/8 BST XIC I:0.1/4 NXB XIC B3:4/0 BND XIO B3:4/1 BST OTE B3:4/0 NXB TON T4:29 1.0 600 600 BND EOR
%   I:0.0/8  AUTO  "Enter Auto Mode" %
%   I:0.1/4  LS3  "Read Bin Size" %
%   B3:4/0  START_CYCLE_TIMER %
%   B3:4/1  RESET_CYCLE_TIMER %
%   T4:29  CYCLE_TIME %
% Rung: 1 %
SOR XIO I:2.0/2 XIC B3:4/0 OSF B3:4/7 B3:4/8 EOR
%   I:2.0/2  PE3  "Gravity Full" %
%   B3:4/0  START_CYCLE_TIMER %
%   B3:4/7  ONE_SHOOT_SET %
%   B3:4/8  SAVE_CYCLE_TIME %
% Rung: 2 %
SOR XIC B3:4/8 BST MOV T4:29.ACC N7:17 NXB OTE B3:4/1 BND EOR
%   B3:4/8  SAVE_CYCLE_TIME %
%   T4:29  CYCLE_TIME %
%   N7:17  LAST_CYCLE_TIME %
%   B3:4/1  RESET_CYCLE_TIMER %
% Rung: 3 %
% *************** Blower and air Nozzle *************** %
SOR XIC B3:3/5 MOV N7:26 T4:20.PRE EOR
%   B3:3/5  SMALL_BIN_SET  "Bin sizzing result" %
%   N7:26  BLOW_DRY_SMALL_BIN %
%   T4:20.PRE  BLOW_OUT_TIME %
% Rung: 4 %
SOR XIC B3:3/6 MOV N7:27 T4:20.PRE EOR
%   B3:3/6  LARGE_BIN_SET  "Bin sizzing result" %
%   N7:27  BLOW_DRY_LARGE_BIN %
%   T4:20.PRE  BLOW_OUT_TIME %
% Rung: 5 %
SOR BST XIC I:0.0/8 XIC B3:0/15 NXB XIO I:0.0/8 XIC B3:3/13 BND XIC I:1.0/2 XIO O:0.0/2 XIO O:0.0/3 LES N7:2 N7:4 BST OTE O:3.0/4 NXB TON T4:20 1.0 1 0 BND EOR
%   I:0.0/8  AUTO  "Enter Auto Mode" %
%   B3:0/15  LATCH_LOWER_AIR %
%   B3:3/13  BLOWER_ENGAGE_TEST  "Touchscreen" %
%   I:1.0/2  LS10  "Brush Out" %
%   O:0.0/2  BRUSH_CW  "VFD run forward" %
%   O:0.0/3  BRUSH_CCW  "VFD run reverse" %
%   N7:2  CRADDLE_DOWN_POSITIO %
%   N7:4  DRYING_POSITION %
%   O:3.0/4  AIR_NOZZLE_IN_ %
%   T4:20  DRYING_TIMER %

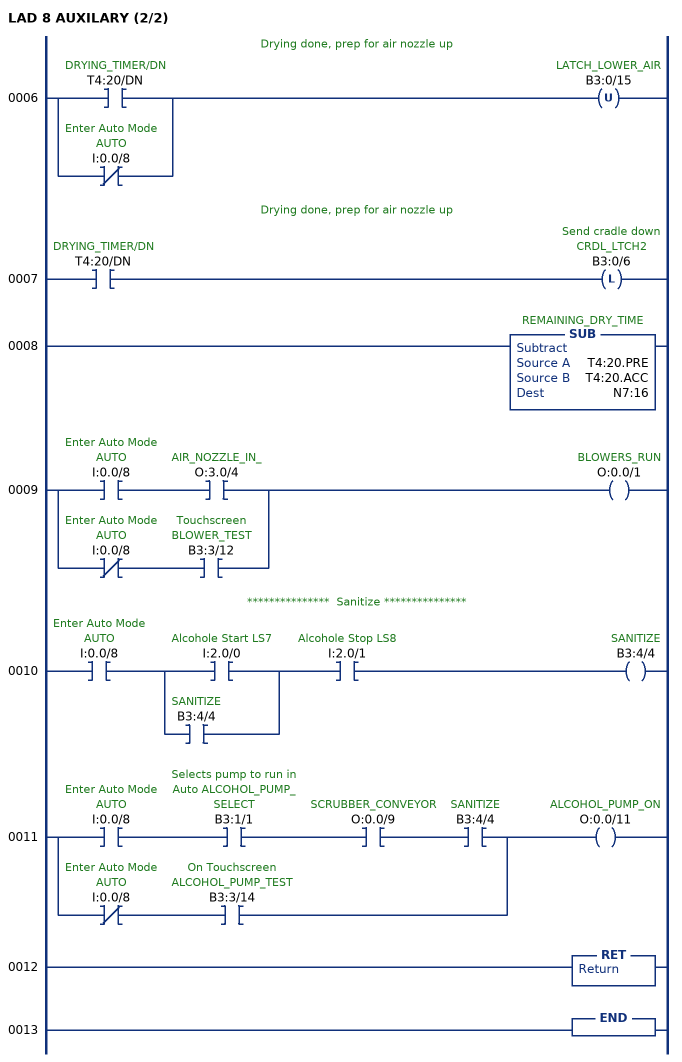
% Rung: 6 %
% Drying done, prep for air nozzle up %
SOR BST XIC T4:20/DN NXB XIO I:0.0/8 BND OTU B3:0/15 EOR
%   T4:20  DRYING_TIMER %
%   I:0.0/8  AUTO  "Enter Auto Mode" %
%   B3:0/15  LATCH_LOWER_AIR %
% Rung: 7 %
% Drying done, prep for air nozzle up %
SOR XIC T4:20/DN OTL B3:0/6 EOR
%   T4:20  DRYING_TIMER %
%   B3:0/6  CRDL_LTCH2  "Send cradle down" %
% Rung: 8 %
SOR SUB T4:20.PRE T4:20.ACC N7:16 EOR
%   T4:20.PRE  BLOW_OUT_TIME %
%   T4:20  DRYING_TIMER %
%   N7:16  REMAINING_DRY_TIME %
% Rung: 9 %
SOR BST XIC I:0.0/8 XIC O:3.0/4 NXB XIO I:0.0/8 XIC B3:3/12 BND OTE O:0.0/1 EOR
%   I:0.0/8  AUTO  "Enter Auto Mode" %
%   O:3.0/4  AIR_NOZZLE_IN_ %
%   B3:3/12  BLOWER_TEST  "Touchscreen" %
%   O:0.0/1  BLOWERS_RUN %
% Rung: 10 %
% ***************  Sanitize *************** %
SOR XIC I:0.0/8 BST XIC I:2.0/0 NXB XIC B3:4/4 BND XIC I:2.0/1 OTE B3:4/4 EOR
%   I:0.0/8  AUTO  "Enter Auto Mode" %
%   I:2.0/0  LS7  "Alcohole Start" %
%   B3:4/4  SANITIZE %
%   I:2.0/1  LS8  "Alcohole Stop" %
% Rung: 11 %
SOR BST XIC I:0.0/8 XIC B3:1/1 XIC O:0.0/9 XIC B3:4/4 NXB XIO I:0.0/8 XIC B3:3/14 BND OTE O:0.0/11 EOR
%   I:0.0/8  AUTO  "Enter Auto Mode" %
%   B3:1/1  ALCOHOL_PUMP_SELECT  "Selects pump to run in Auto" %
%   O:0.0/9  SCRUBBER_CONVEYOR %
%   B3:4/4  SANITIZE %
%   B3:3/14  ALCOHOL_PUMP_TEST  "On Touchscreen" %
%   O:0.0/11  ALCOHOL_PUMP_ON %
% Rung: 12 %
SOR RET EOR
% Rung: 13 %
SOR END EOR

LADDER 9 "FAULTS"
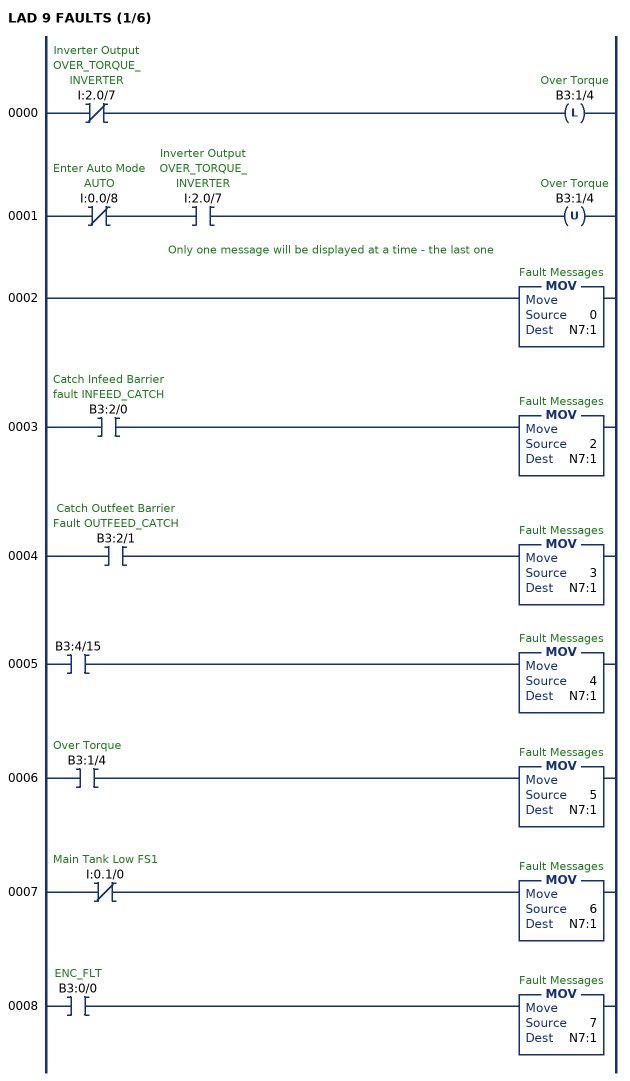
% Rung: 0 %
SOR XIO I:2.0/7 OTL B3:1/4 EOR
%   I:2.0/7  OVER_TORQUE_INVERTER  "Inverter Output" %
%   B3:1/4  "Over Torque" %
% Rung: 1 %
SOR XIO I:0.0/8 XIC I:2.0/7 OTU B3:1/4 EOR
%   I:0.0/8  AUTO  "Enter Auto Mode" %
%   I:2.0/7  OVER_TORQUE_INVERTER  "Inverter Output" %
%   B3:1/4  "Over Torque" %
% Rung: 2 %
% Only one message will be displayed at a time - the last one %
SOR MOV 0 N7:1 EOR
%   N7:1  "Fault Messages" %
% Rung: 3 %
SOR XIC B3:2/0 MOV 2 N7:1 EOR
%   B3:2/0  INFEED_CATCH  "Catch Infeed Barrier fault" %
%   N7:1  "Fault Messages" %
% Rung: 4 %
SOR XIC B3:2/1 MOV 3 N7:1 EOR
%   B3:2/1  OUTFEED_CATCH  "Catch Outfeet Barrier Fault" %
%   N7:1  "Fault Messages" %
% Rung: 5 %
SOR XIC B3:4/15 MOV 4 N7:1 EOR
%   N7:1  "Fault Messages" %
% Rung: 6 %
SOR XIC B3:1/4 MOV 5 N7:1 EOR
%   B3:1/4  "Over Torque" %
%   N7:1  "Fault Messages" %
% Rung: 7 %
SOR XIO I:0.1/0 MOV 6 N7:1 EOR
%   I:0.1/0  FS1  "Main Tank Low" %
%   N7:1  "Fault Messages" %
% Rung: 8 %
SOR XIC B3:0/0 MOV 7 N7:1 EOR
%   B3:0/0  ENC_FLT %
%   N7:1  "Fault Messages" %

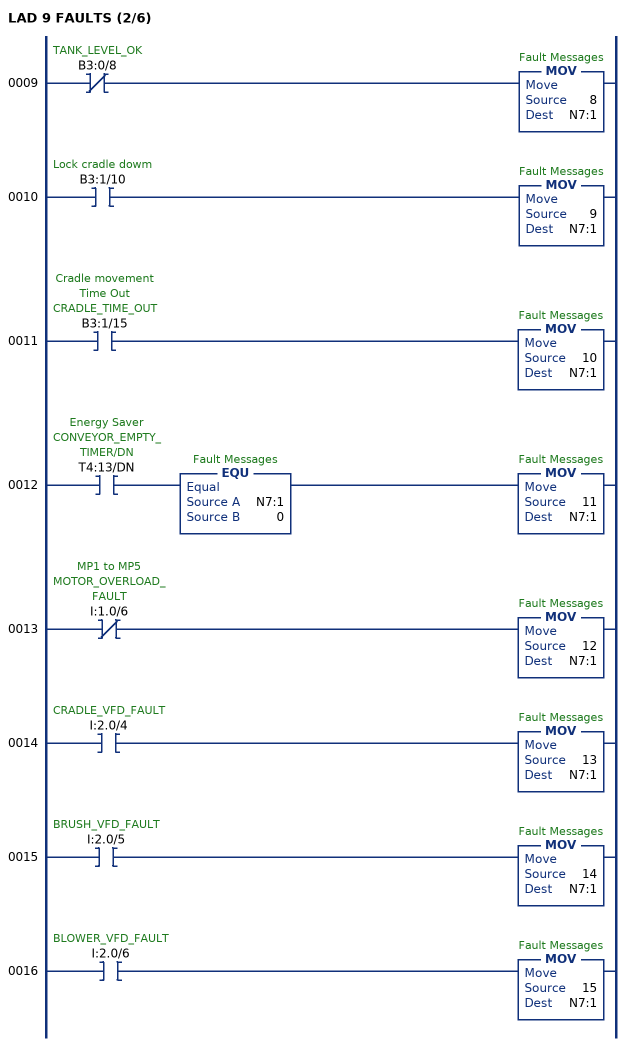
% Rung: 9 %
SOR XIO B3:0/8 MOV 8 N7:1 EOR
%   B3:0/8  TANK_LEVEL_OK %
%   N7:1  "Fault Messages" %
% Rung: 10 %
SOR XIC B3:1/10 MOV 9 N7:1 EOR
%   B3:1/10  "Lock cradle dowm" %
%   N7:1  "Fault Messages" %
% Rung: 11 %
SOR XIC B3:1/15 MOV 10 N7:1 EOR
%   B3:1/15  CRADLE_TIME_OUT  "Cradle movement Time Out" %
%   N7:1  "Fault Messages" %
% Rung: 12 %
SOR XIC T4:13/DN EQU N7:1 0 MOV 11 N7:1 EOR
%   T4:13  CONVEYOR_EMPTY_TIMER  "Energy Saver" %
%   N7:1  "Fault Messages" %
% Rung: 13 %
SOR XIO I:1.0/6 MOV 12 N7:1 EOR
%   I:1.0/6  MOTOR_OVERLOAD_FAULT  "MP1 to MP5" %
%   N7:1  "Fault Messages" %
% Rung: 14 %
SOR XIC I:2.0/4 MOV 13 N7:1 EOR
%   I:2.0/4  CRADLE_VFD_FAULT %
%   N7:1  "Fault Messages" %
% Rung: 15 %
SOR XIC I:2.0/5 MOV 14 N7:1 EOR
%   I:2.0/5  BRUSH_VFD_FAULT %
%   N7:1  "Fault Messages" %
% Rung: 16 %
SOR XIC I:2.0/6 MOV 15 N7:1 EOR
%   I:2.0/6  BLOWER_VFD_FAULT %
%   N7:1  "Fault Messages" %

